FUNCTION_BLOCK FB_BatchJobContainerCreator IMPLEMENTS I_TaskCreator
VAR_INPUT
END_VAR
VAR_OUTPUT
END_VAR
VAR
END_VAR

METHOD create_future : I_Future
VAR_INPUT
	future_name :STRING;
END_VAR
VAR
	_p_future : POINTER TO FB_BatchJobContainer;
END_VAR
_p_future := __NEW(FB_BatchJobContainer);
_p_future^.future_name := future_name;
create_future := _p_future^;
END_METHOD

{warning 'add method implementation '}
METHOD destroy_future : I_Future
VAR_INPUT
	future	: I_Future;
END_VAR
VAR
	_p_future : POINTER TO FB_BatchJobContainer;
END_VAR
IF __QUERYPOINTER(future, _p_future) THEN
	__DELETE(_p_future);
	IF _p_future = 0  THEN
		destroy_future := 0;
	END_IF
END_IF
END_METHOD

END_FUNCTION_BLOCK

(* stored: Version 1.1.0.1, ProductVersion 3.1.4026.17
   POU FB_BatchJobContainerCreator: Id {cc44dec9-caab-4c2a-8bde-99d401648394}, SpecialFunc None
   Method create_future: Id {2a5ce7c8-44bb-4ea8-88ae-9f8a9b48cc13}
   Method destroy_future: Id {af7c8340-e0c5-499c-81af-0833eba2fa7d} *)
